// TIA Portal V17 export
// export: Created 2024-09-03T21:54:57.8693809Z, ExportSetting WithDefaults, DisplayName Totally Integrated Automation Portal, DisplayVersion V17 Update 7, DisplayName TIA Portal Openness, DisplayVersion V17 Update 7, DisplayName TIA Portal Version Control Interface, DisplayVersion V17, DisplayName SINAMICS Startdrive Advanced, DisplayVersion V17 SP2, DisplayName SINAMICS Startdrive G110M, G120, G120C, G120D, G120P, G115D, DisplayVersion V17 SP2, DisplayName SINAMICS Startdrive G130, G150, S120, S150, SINAMICS MV, S210, DisplayVersion V17 SP2, DisplayName STEP 7 Professional, DisplayVersion V17 Update 7, DisplayName STEP 7 Safety, DisplayVersion V17 Update 6, DisplayName WinCC Advanced / Unified PC, DisplayVersion V17 Update 7
FUNCTION_BLOCK "sq_carousel_main"   // FB70, GRAPH
VERSION : 0.1
// stored: AcknowledgeErrorsRequired true, AutoNumber true, GraphVersion 6.0, InitialValuesAcquisition false, IsIECCheckEnabled false, LanguageInNetworks LAD, LockOperatingMode false, PermanentILProcessingInMANMode false, SetENOAutomatically false, SkipSteps false, UDAEnableTagReadback false, WithAlarmHandling true
   // inherited from GRAPH_BASE
   VAR
      OFF_SQ_BASE : Bool;
   END_VAR
   VAR_INPUT
      OFF_SQ { ExternalAccessible := 'False'; ExternalVisible := 'False'; ExternalWritable := 'False'} : Bool := false;   // Turn sequence off
      INIT_SQ { ExternalAccessible := 'False'; ExternalVisible := 'False'; ExternalWritable := 'False'} : Bool := false;   // Set sequence to initial state
      ACK_EF { ExternalAccessible := 'False'; ExternalVisible := 'False'; ExternalWritable := 'False'} : Bool := false;   // Acknowledge all errors and faults
      S_PREV { ExternalAccessible := 'False'; ExternalVisible := 'False'; ExternalWritable := 'False'} : Bool := false;   // Output previous step in parameter S_NO
      S_NEXT { ExternalAccessible := 'False'; ExternalVisible := 'False'; ExternalWritable := 'False'} : Bool := false;   // Indicate next step in parameter S_NO
      SW_AUTO { ExternalAccessible := 'False'; ExternalVisible := 'False'; ExternalWritable := 'False'} : Bool := false;   // Automatic mode
      SW_TAP { ExternalAccessible := 'False'; ExternalVisible := 'False'; ExternalWritable := 'False'} : Bool := false;   // Semiautomatic/switch with transition
      SW_TOP { ExternalAccessible := 'False'; ExternalVisible := 'False'; ExternalWritable := 'False'} : Bool := false;   // Semiautomatic/ignore transition
      SW_MAN { ExternalAccessible := 'False'; ExternalVisible := 'False'; ExternalWritable := 'False'} : Bool := false;   // Manual mode
      S_SEL { ExternalAccessible := 'False'; ExternalVisible := 'False'; ExternalWritable := 'False'} : Int := 0;   // Select step to be output to S_NO
      S_ON { ExternalAccessible := 'False'; ExternalVisible := 'False'; ExternalWritable := 'False'} : Bool := false;   // Activate step indicated in S_NO
      S_OFF { ExternalAccessible := 'False'; ExternalVisible := 'False'; ExternalWritable := 'False'} : Bool := false;   // Deactivate step indicated S_NO
      T_PUSH { ExternalAccessible := 'False'; ExternalVisible := 'False'; ExternalWritable := 'False'} : Bool := false;   // Enable transition to switch in semi automatic mode
   END_VAR
   VAR_OUTPUT
      S_NO { ExternalAccessible := 'False'; ExternalVisible := 'False'; ExternalWritable := 'False'} : Int := 0;   // Step number
      S_MORE { ExternalAccessible := 'False'; ExternalVisible := 'False'; ExternalWritable := 'False'} : Bool := false;   // More steps are available and can be shown in S_NO
      S_ACTIVE { ExternalAccessible := 'False'; ExternalVisible := 'False'; ExternalWritable := 'False'} : Bool := false;   // Step indicated in S_NO is active
      ERR_FLT { ExternalAccessible := 'False'; ExternalVisible := 'False'; ExternalWritable := 'False'} : Bool := false;   // Interlock or supervision group error
      AUTO_ON { ExternalAccessible := 'False'; ExternalVisible := 'False'; ExternalWritable := 'False'} : Bool := false;   // Automatic mode is active
      TAP_ON { ExternalAccessible := 'False'; ExternalVisible := 'False'; ExternalWritable := 'False'} : Bool := false;   // Semiautomatic mode/step with transition enabled
      TOP_ON { ExternalAccessible := 'False'; ExternalVisible := 'False'; ExternalWritable := 'False'} : Bool := false;   // Semiautomatic mode/ignore transition enabled
      MAN_ON { ExternalAccessible := 'False'; ExternalVisible := 'False'; ExternalWritable := 'False'} : Bool := false;   // Manual mode is active
   END_VAR
   VAR
      dummy : Bool;
      start : Bool;
      base : Bool;
   END_VAR
BEGIN
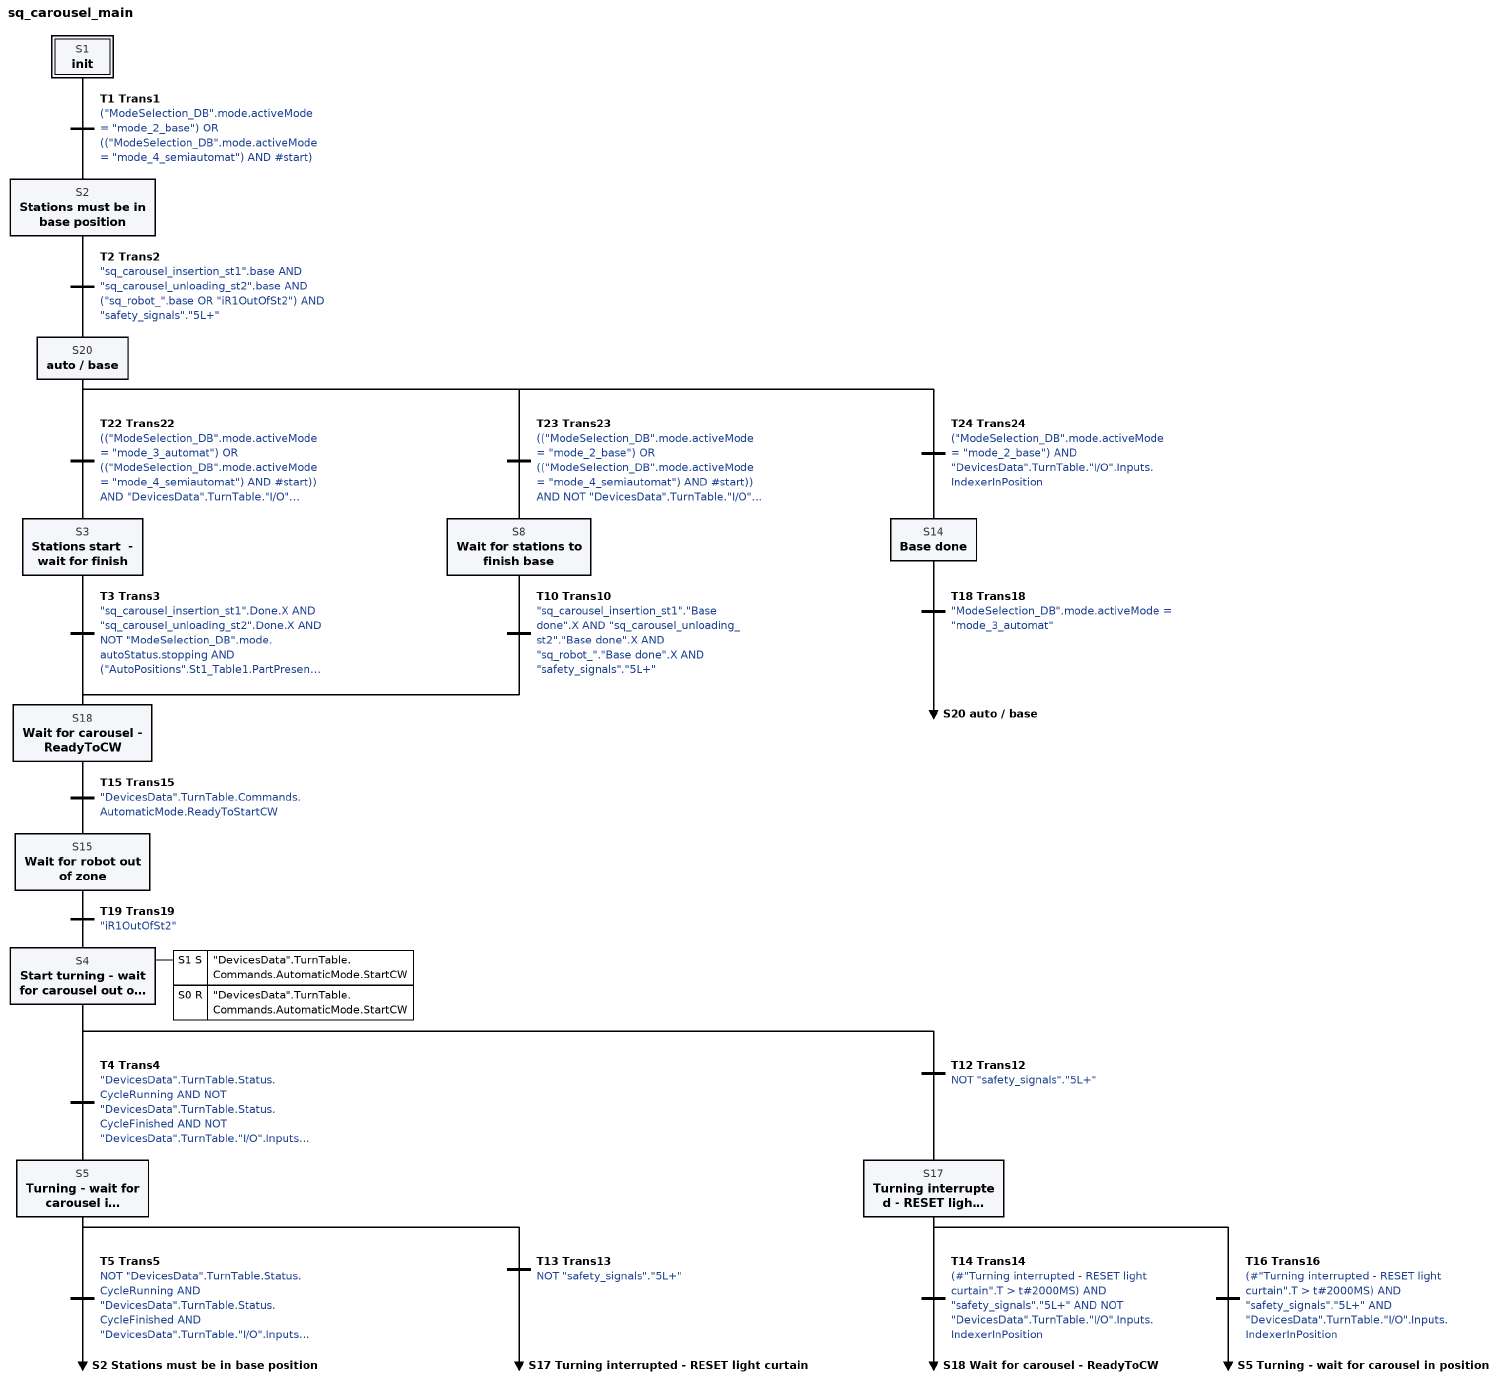
   // permanent pre-instructions
   NETWORK 1
      #base := "iTurnTableIndexerInPosition";

   // sequencer 1
   INITIAL_STEP init:   // S1, max time T#10S, warning time T#7S
   END_STEP
   TRANSITION Trans1 FROM init TO "Stations must be in base position"   // T1
      := ("ModeSelection_DB".mode.activeMode = "mode_2_base") OR (("ModeSelection_DB".mode.activeMode = "mode_4_semiautomat") AND #start);
   END_TRANSITION
   STEP "Stations must be in base position":   // S2, max time T#10S, warning time T#7S
      supervision V := #"Stations must be in base position".T > #"Stations must be in base position".T_MAX;
   END_STEP
   TRANSITION Trans2 FROM "Stations must be in base position" TO "auto / base"   // T2
      := "sq_carousel_insertion_st1".base AND "sq_carousel_unloading_st2".base AND ("sq_robot_".base OR "iR1OutOfSt2") AND "safety_signals"."5L+";
   END_TRANSITION
   STEP "Stations start  - wait for finish":   // S3, max time T#10S, warning time T#7S
   END_STEP
   TRANSITION Trans3 FROM "Stations start  - wait for finish" TO "Wait for carousel - ReadyToCW"   // T3
      := "sq_carousel_insertion_st1".Done.X AND "sq_carousel_unloading_st2".Done.X AND NOT "ModeSelection_DB".mode.autoStatus.stopping AND ("AutoPositions".St1_Table1.PartPresent OR "AutoPositions".St2_Table2.PartPresent OR NOT "ModeSelection_DB".mode.autoStatus.emptying) AND "safety_signals"."5L+";
   END_TRANSITION
   STEP "Start turning - wait for carousel out of position":   // S4, max time T#10S, warning time T#7S
      supervision V := #"Start turning - wait for carousel out of position".T > #"Start turning - wait for carousel out of position".T_MAX;
          S1  S    "DevicesData".TurnTable.Commands.AutomaticMode.StartCW
          S0  R    "DevicesData".TurnTable.Commands.AutomaticMode.StartCW
   END_STEP
   TRANSITION Trans4 FROM "Start turning - wait for carousel out of position" TO "Turning - wait for carousel in position"   // T4
      := "DevicesData".TurnTable.Status.CycleRunning AND NOT "DevicesData".TurnTable.Status.CycleFinished AND NOT "DevicesData".TurnTable."I/O".Inputs.IndexerInPosition;
   END_TRANSITION
   TRANSITION Trans12 FROM "Start turning - wait for carousel out of position" TO "Turning interrupted - RESET light curtain"   // T12
      := NOT "safety_signals"."5L+";
   END_TRANSITION
   STEP "Turning - wait for carousel in position":   // S5, max time T#10S, warning time T#7S
      supervision V := #"Turning - wait for carousel in position".T > #"Turning - wait for carousel in position".T_MAX;
   END_STEP
   TRANSITION Trans5 FROM "Turning - wait for carousel in position" TO "Stations must be in base position"   // T5, jump
      := NOT "DevicesData".TurnTable.Status.CycleRunning AND "DevicesData".TurnTable.Status.CycleFinished AND "DevicesData".TurnTable."I/O".Inputs.IndexerInPosition;
   END_TRANSITION
   TRANSITION Trans13 FROM "Turning - wait for carousel in position" TO "Turning interrupted - RESET light curtain"   // T13, jump
      := NOT "safety_signals"."5L+";
   END_TRANSITION
   STEP "Turning interrupted - RESET light curtain":   // S17, max time T#10S, warning time T#7S
   END_STEP
   TRANSITION Trans14 FROM "Turning interrupted - RESET light curtain" TO "Wait for carousel - ReadyToCW"   // T14, jump
      := (#"Turning interrupted - RESET light curtain".T > t#2000MS) AND "safety_signals"."5L+" AND NOT "DevicesData".TurnTable."I/O".Inputs.IndexerInPosition;
   END_TRANSITION
   TRANSITION Trans16 FROM "Turning interrupted - RESET light curtain" TO "Turning - wait for carousel in position"   // T16, jump
      := (#"Turning interrupted - RESET light curtain".T > t#2000MS) AND "safety_signals"."5L+" AND "DevicesData".TurnTable."I/O".Inputs.IndexerInPosition;
   END_TRANSITION
   STEP "Wait for carousel - ReadyToCW":   // S18, max time T#10S, warning time T#7S
      supervision V := #"Wait for carousel - ReadyToCW".T > #"Wait for carousel - ReadyToCW".T_MAX;
   END_STEP
   TRANSITION Trans15 FROM "Wait for carousel - ReadyToCW" TO "Wait for robot out of zone"   // T15
      := "DevicesData".TurnTable.Commands.AutomaticMode.ReadyToStartCW;
   END_TRANSITION
   STEP "Wait for stations to finish base":   // S8, max time T#10S, warning time T#7S
   END_STEP
   TRANSITION Trans10 FROM "Wait for stations to finish base" TO "Wait for carousel - ReadyToCW"   // T10
      := "sq_carousel_insertion_st1"."Base done".X AND "sq_carousel_unloading_st2"."Base done".X AND "sq_robot_"."Base done".X AND "safety_signals"."5L+";
   END_TRANSITION
   STEP "auto / base":   // S20, max time T#10S, warning time T#7S
   END_STEP
   TRANSITION Trans22 FROM "auto / base" TO "Stations start  - wait for finish"   // T22
      := (("ModeSelection_DB".mode.activeMode = "mode_3_automat") OR (("ModeSelection_DB".mode.activeMode = "mode_4_semiautomat") AND #start)) AND "DevicesData".TurnTable."I/O".Inputs.IndexerInPosition;
   END_TRANSITION
   TRANSITION Trans23 FROM "auto / base" TO "Wait for stations to finish base"   // T23
      := (("ModeSelection_DB".mode.activeMode = "mode_2_base") OR (("ModeSelection_DB".mode.activeMode = "mode_4_semiautomat") AND #start)) AND NOT "DevicesData".TurnTable."I/O".Inputs.IndexerInPosition;
   END_TRANSITION
   TRANSITION Trans24 FROM "auto / base" TO "Base done"   // T24
      := ("ModeSelection_DB".mode.activeMode = "mode_2_base") AND "DevicesData".TurnTable."I/O".Inputs.IndexerInPosition;
   END_TRANSITION
   STEP "Base done":   // S14, max time T#10S, warning time T#7S
   END_STEP
   TRANSITION Trans18 FROM "Base done" TO "auto / base"   // T18, jump
      := "ModeSelection_DB".mode.activeMode = "mode_3_automat";
   END_TRANSITION
   STEP "Wait for robot out of zone":   // S15, max time T#10S, warning time T#7S
      supervision V := #"Wait for robot out of zone".T > #"Wait for robot out of zone".T_MAX;
   END_STEP
   TRANSITION Trans19 FROM "Wait for robot out of zone" TO "Start turning - wait for carousel out of position"   // T19
      := "iR1OutOfSt2";
   END_TRANSITION
END_FUNCTION_BLOCK
